// SIMATIC S7-200 project (STEP 7-Micro/WIN), CPU 226 REL 02.01

ORGANIZATION_BLOCK OB:OB1
TITLE=2008.01.10更改
BEGIN
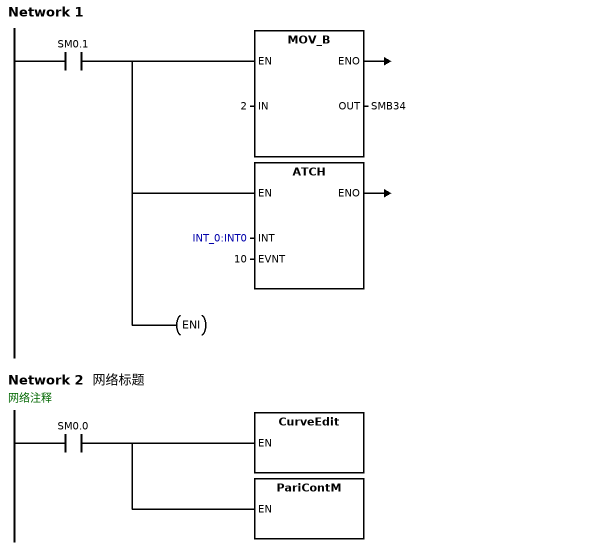
Network 1
LD     SM0.1
MOVB   2, SMB34
ATCH   INT_0:INT0, 10
ENI
Network 2 // 网络标题
// 网络注释
LD     SM0.0
CALL   CurveEdit:SBR61
CALL   PariContM:SBR62
END_ORGANIZATION_BLOCK

// SBR61: protected block, not included

// SBR62: protected block, not included

// SBR63: protected block, not included

INTERRUPT_BLOCK INT_0:INT0
TITLE=中断程序注释
BEGIN
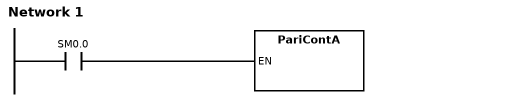
Network 1
LD     SM0.0
CALL   PariContA:SBR63
END_INTERRUPT_BLOCK
